FUNCTION_BLOCK ASSEMBLE_AL_FROM_AB (* this Function combines the 8 AB (BYTE) adapters to a AL (LWORD) *)
  (* Standard: 61499-2; Description: Copyright (c) 2026 Meisterschulen am Ostbahnhof SPDX-License-Identifier: EPL-2.0 *)
  (* Version 1.0, 2026-05-16, Franz Höpfinger, Meisterschulen am Ostbahnhof, initial API and implementation and/or initial documentation *)
  PACKAGE adapter::assembling;
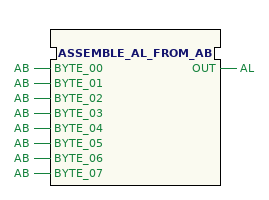
  SOCKETS
    BYTE_00 : adapter::types::unidirectional::AB; (* Byte 0 *)
    BYTE_01 : adapter::types::unidirectional::AB; (* Byte 1 *)
    BYTE_02 : adapter::types::unidirectional::AB; (* Byte 2 *)
    BYTE_03 : adapter::types::unidirectional::AB; (* Byte 3 *)
    BYTE_04 : adapter::types::unidirectional::AB; (* Byte 4 *)
    BYTE_05 : adapter::types::unidirectional::AB; (* Byte 5 *)
    BYTE_06 : adapter::types::unidirectional::AB; (* Byte 6 *)
    BYTE_07 : adapter::types::unidirectional::AB; (* Byte 7 *)
  END_SOCKETS
  PLUGS
    OUT : adapter::types::unidirectional::AL; (* LWORD Output *)
  END_PLUGS
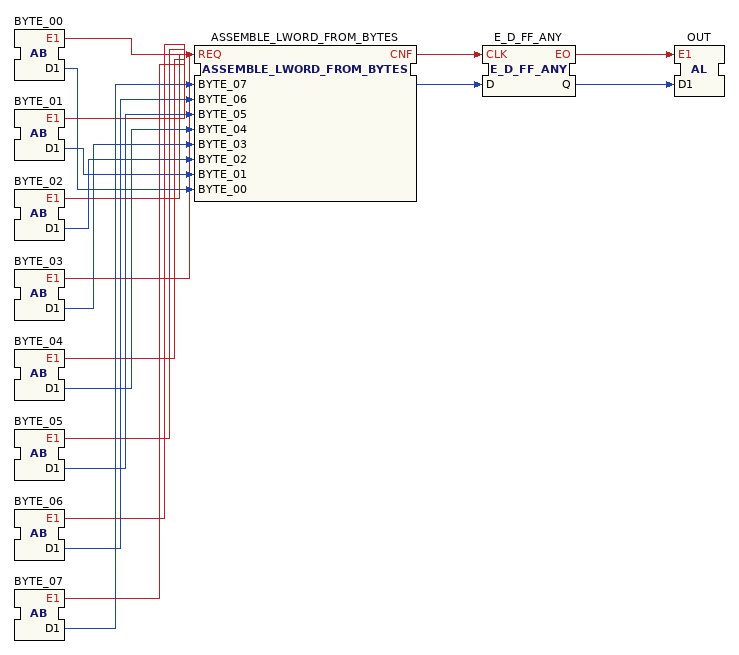
  FBS
    ASSEMBLE_LWORD_FROM_BYTES : eclipse4diac::utils::assembling::ASSEMBLE_LWORD_FROM_BYTES;
    E_D_FF_ANY : iec61499::events::E_D_FF_ANY;
  END_FBS
  EVENT_CONNECTIONS
    BYTE_00.E1 TO ASSEMBLE_LWORD_FROM_BYTES.REQ;
    BYTE_01.E1 TO ASSEMBLE_LWORD_FROM_BYTES.REQ;
    BYTE_02.E1 TO ASSEMBLE_LWORD_FROM_BYTES.REQ;
    BYTE_03.E1 TO ASSEMBLE_LWORD_FROM_BYTES.REQ;
    BYTE_04.E1 TO ASSEMBLE_LWORD_FROM_BYTES.REQ;
    BYTE_05.E1 TO ASSEMBLE_LWORD_FROM_BYTES.REQ;
    BYTE_06.E1 TO ASSEMBLE_LWORD_FROM_BYTES.REQ;
    BYTE_07.E1 TO ASSEMBLE_LWORD_FROM_BYTES.REQ;
    ASSEMBLE_LWORD_FROM_BYTES.CNF TO E_D_FF_ANY.CLK;
    E_D_FF_ANY.EO TO OUT.E1;
  END_CONNECTIONS
  DATA_CONNECTIONS
    ASSEMBLE_LWORD_FROM_BYTES. TO E_D_FF_ANY.D;
    E_D_FF_ANY.Q TO OUT.D1;
    BYTE_07.D1 TO ASSEMBLE_LWORD_FROM_BYTES.BYTE_07;
    BYTE_06.D1 TO ASSEMBLE_LWORD_FROM_BYTES.BYTE_06;
    BYTE_05.D1 TO ASSEMBLE_LWORD_FROM_BYTES.BYTE_05;
    BYTE_04.D1 TO ASSEMBLE_LWORD_FROM_BYTES.BYTE_04;
    BYTE_03.D1 TO ASSEMBLE_LWORD_FROM_BYTES.BYTE_03;
    BYTE_02.D1 TO ASSEMBLE_LWORD_FROM_BYTES.BYTE_02;
    BYTE_01.D1 TO ASSEMBLE_LWORD_FROM_BYTES.BYTE_01;
    BYTE_00.D1 TO ASSEMBLE_LWORD_FROM_BYTES.BYTE_00;
  END_CONNECTIONS
END_FUNCTION_BLOCK
